FUNCTION_BLOCK MIXER_V1 (* Mixer Communication Block V1 *)
  (* Standard: 61499-2 *)
  (* Version 1.0, 2023-08-25, ADMIN *)
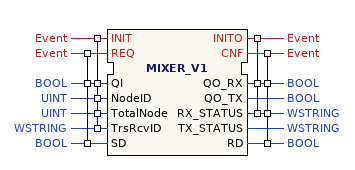
  EVENT_INPUT
    INIT WITH QI, NodeID, TotalNode, TrsRcvID; (* Initialization Request *)
    REQ WITH QI, SD; (* Normal Execution Request *)
  END_EVENT
  EVENT_OUTPUT
    INITO WITH QO_RX, RX_STATUS; (* Initialization Confirm *)
    CNF WITH QO_RX, RX_STATUS, RD; (* Execution Confirmation *)
  END_EVENT
  VAR_INPUT
    QI : BOOL;
    NodeID : UINT;
    TotalNode : UINT;
    TrsRcvID : WSTRING;
    SD : BOOL;
  END_VAR
  VAR_OUTPUT
    QO_RX : BOOL;
    QO_TX : BOOL;
    RX_STATUS : WSTRING;
    TX_STATUS : WSTRING;
    RD : BOOL;
  END_VAR
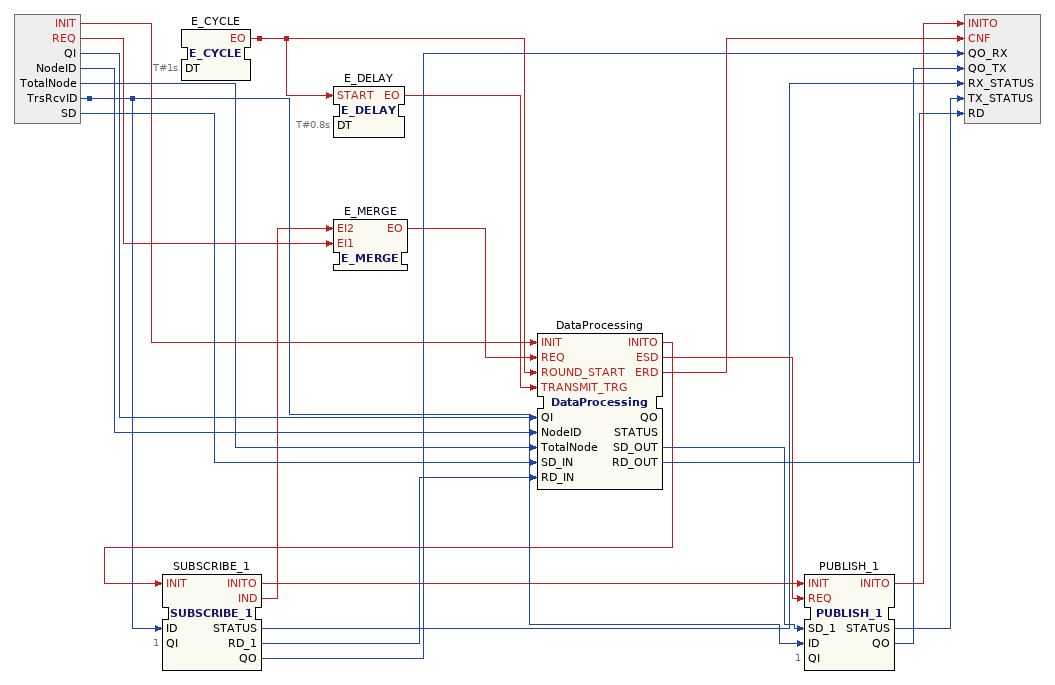
  FBS
    E_CYCLE : E_CYCLE(DT := T#1s);
    E_DELAY : E_DELAY(DT := T#0.8s);
    PUBLISH_1 : PUBLISH_1(QI := 1);
    SUBSCRIBE_1 : SUBSCRIBE_1(QI := 1);
    E_MERGE : E_MERGE;
    DataProcessing : DataProcessing;
  END_FBS
  EVENT_CONNECTIONS
    E_CYCLE.EO TO E_DELAY.START;
    SUBSCRIBE_1.INITO TO PUBLISH_1.INIT;
    PUBLISH_1.INITO TO INITO;
    SUBSCRIBE_1.IND TO E_MERGE.EI2;
    REQ TO E_MERGE.EI1;
    DataProcessing.INITO TO SUBSCRIBE_1.INIT;
    DataProcessing.ESD TO PUBLISH_1.REQ;
    DataProcessing.ERD TO CNF;
    INIT TO DataProcessing.INIT;
    E_MERGE.EO TO DataProcessing.REQ;
    E_CYCLE.EO TO DataProcessing.ROUND_START;
    E_DELAY.EO TO DataProcessing.TRANSMIT_TRG;
  END_CONNECTIONS
  DATA_CONNECTIONS
    SUBSCRIBE_1.STATUS TO RX_STATUS;
    PUBLISH_1.STATUS TO TX_STATUS;
    DataProcessing.SD_OUT TO PUBLISH_1.SD_1;
    DataProcessing.RD_OUT TO RD;
    QI TO DataProcessing.QI;
    SD TO DataProcessing.SD_IN;
    SUBSCRIBE_1.RD_1 TO DataProcessing.RD_IN;
    NodeID TO DataProcessing.NodeID;
    TotalNode TO DataProcessing.TotalNode;
    SUBSCRIBE_1.QO TO QO_RX;
    PUBLISH_1.QO TO QO_TX;
    TrsRcvID TO SUBSCRIBE_1.ID;
    TrsRcvID TO PUBLISH_1.ID;
  END_CONNECTIONS
END_FUNCTION_BLOCK
